PROGRAM MAIN
VAR
	// trigger command execution for Postman-Echo samples
	bGet, bPost, bPut, bHeaderAuth 	: BOOL;

	fbHttpClientPostman				: FB_IotHttpClient :=(sHostName:= '127.0.0.1' , // 'postman-echo.com',
								  	bKeepAlive:=FALSE, tConnectionTimeout:=T#30S);
								//'postman-echo.com'
	fbHttpGet						: FB_TestHTTP_Get;
	fbHttpPost						: FB_TestHTTP_Post;
	fbHttpPut						: FB_TestHTTP_Put;
	fbHttpHeaderAuth				: FB_TestHTTP_HeaderAuth;

END_VAR

// init client parameters at startup
IF NOT fbHttpClientPostman.bConfigured THEN 
	fbHttpClientPostman.nHostPort:=  1234;  // 80; //
	
END_IF

IF fbHttpClientPostman.bConfigured THEN 
	fbHttpGet(bSend:=bGet, fbClient:=fbHttpClientPostman);
	fbHttpPost(bSend:=bPost, fbClient:=fbHttpClientPostman);
	fbHttpPut(bSend:=bPut, fbClient:=fbHttpClientPostman);
	fbHttpHeaderAuth(bSend:=bHeaderAuth, fbClient:=fbHttpClientPostman);
END_IF 

fbHttpClientPostman.Execute();

END_PROGRAM

(* stored: Version 1.1.0.1, ProductVersion 3.1.4024.12
   POU MAIN: Id {b37e2b32-48ef-44fd-8d39-b46780530972}, SpecialFunc None *)
